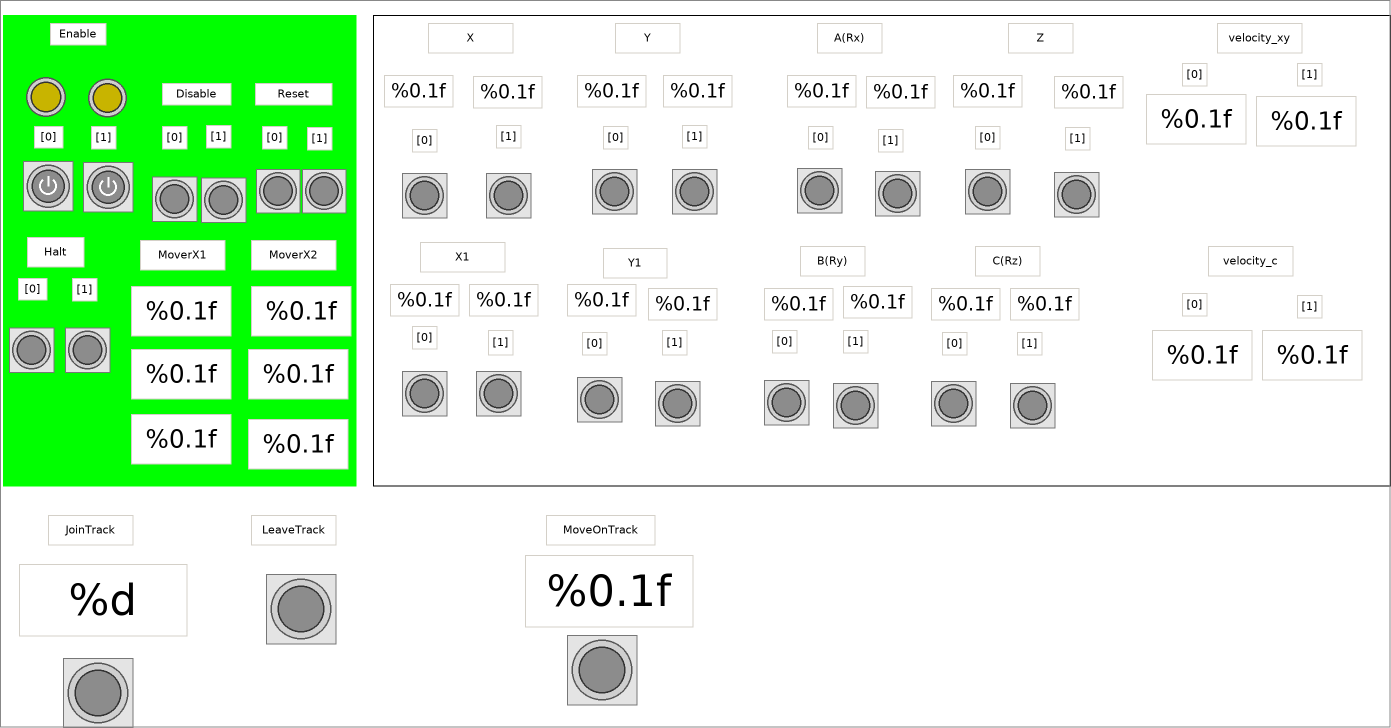
VISUALIZATION Visualization  // 1391x728
    Rectangle (373,15 1018x471)
    Rectangle (3,15 353x471)
    PowerSwitch (23,158 50x56), tooltip "Enable", variable: MAIN.enableM[0], behaviour: TOGGLE, style: Switch-PowerSwitch-Gray
    PushSwitch (152,159 45x80), tooltip "disable", variable: MAIN.disableM[0], behaviour: TAP, style: Switch-PushSwitch-Gray
    Lamp1 (23,64 46x66), variable: MAIN.Xpfeedback[0][0].Done, style: Lamp-Lamp1-Yellow
    PushSwitchLed (402,161 45x69), tooltip "movex", variable: MAIN.moveXM[0], behaviour: TOGGLE, style: Switch-PushSwitchLed-Gray
    Textfield (384,75 69x32), "%0.1f", text variable: MAIN.positionTargetX[0]
        OnMouseClick: write the text variable via Default, min 60, max 660
    Textfield (428,23 85x30), "X"
    Textfield (577,75 69x32), "%0.1f", text variable: MAIN.positionTargetY[0]
        OnMouseClick: write the text variable via Default, min 60, max 420
    Textfield (615,23 65x30), "Y"
    PushSwitchLed (592,160 45x63), tooltip "moveY", variable: MAIN.moveYM[0], behaviour: TOGGLE, style: Switch-PushSwitchLed-Gray
    Textfield (420,242 85x30), "X1"
    Textfield (603,248 64x30), "Y1"
    PushSwitchLed (402,359 45x69), tooltip "movex1", variable: MAIN.moveX1M[0], behaviour: TOGGLE, style: Switch-PushSwitchLed-Gray
    PushSwitchLed (577,365 45x69), tooltip "moveY1", variable: MAIN.moveY1M[0], behaviour: TOGGLE, style: Switch-PushSwitchLed-Gray
    Textfield (390,284 69x32), "%0.1f", text variable: MAIN.positionTargetX1[0]
        OnMouseClick: write the text variable via Default, min 60, max 660
    Textfield (567,284 69x32), "%0.1f", text variable: MAIN.positionTargetY1[0]
        OnMouseClick: write the text variable via Default, min 60, max 420
    Textfield (1146,94 100x50), "%0.1f", text variable: MAIN.velocity_xy[0]
        OnMouseClick: write the text variable via Default, min 1, max 2000
    Textfield (1217,23 85x30), "velocity_xy"
    Textfield (817,23 65x30), "A(Rx)"
    Textfield (787,75 69x32), "%0.1f", text variable: MAIN.positionTargetA[0]
        OnMouseClick: write the text variable via Default, min -5, max 5
    PushSwitchLed (797,159 45x63), tooltip "moveA", variable: MAIN.moveAM[0], behaviour: TOGGLE, style: Switch-PushSwitchLed-Gray
    Textfield (800,246 65x30), "B(Ry)"
    Textfield (764,288 69x32), "%0.1f", text variable: MAIN.positionTargetB[0]
        OnMouseClick: write the text variable via Default, min -5, max 5
    PushSwitchLed (764,368 45x69), tooltip "moveB", variable: MAIN.moveBM[0], behaviour: TOGGLE, style: Switch-PushSwitchLed-Gray
    Textfield (1008,23 65x30), "Z"
    Textfield (953,75 69x32), "%0.1f", text variable: MAIN.positionTargetZ[0]
        OnMouseClick: write the text variable via Default, min 2, max 5
    PushSwitchLed (965,160 45x63), tooltip "moveZ", variable: MAIN.moveZM[0], behaviour: TOGGLE, style: Switch-PushSwitchLed-Gray
    Textfield (975,246 65x30), "C(Rz)"
    Textfield (931,288 69x32), "%0.1f", text variable: MAIN.positionTargetC[0]
        OnMouseClick: write the text variable via Default
    PushSwitchLed (931,369 45x69), tooltip "moveC", variable: MAIN.moveCM[0], behaviour: TOGGLE, style: Switch-PushSwitchLed-Gray
    Textfield (1208,246 85x30), "velocity_c"
    Textfield (1152,330 100x50), "%0.1f", text variable: MAIN.velocity_c[0]
        OnMouseClick: write the text variable via Default, min 1, max 7000
    Textfield (131,286 100x50), "%0.1f", text variable: MAIN.Xpmover[0].MCTOPLC.ACT.ActPos.x
    Textfield (131,349 100x50), "%0.1f", text variable: MAIN.Xpmover[0].MCTOPLC.ACT.ActPos.y
    Textfield (131,414 100x50), "%0.1f", text variable: MAIN.Xpmover[0].MCTOPLC.ACT.ActPos.c
    Textfield (140,240 85x30), "MoverX1"
    PushSwitch (63,658 70x70), variable: MAIN.JoinTrack[0], behaviour: TOGGLE, style: Switch-PushSwitch-Gray
    PushSwitch (266,574 70x70), variable: MAIN.LeaveTrack[0], behaviour: TOGGLE, style: Switch-PushSwitch-Gray
    PushSwitch (567,635 70x70), variable: MAIN.MoveOnTrack[0], behaviour: TOGGLE, style: Switch-PushSwitch-Gray
    Textfield (48,515 85x30), "JoinTrack"
    Textfield (251,515 85x30), "LeaveTrack"
    Textfield (546,515 109x30), "MoveOnTrack"
    Textfield (19,564 168x72), "%d", text variable: MAIN.numberTrack[0]
        OnMouseClick: write the text variable via Default, min 0
    Textfield (525,555 168x72), "%0.1f", text variable: MAIN.distanceTrack[0]
        OnMouseClick: write the text variable via Default
    PushSwitch (256,160 44x62), variable: MAIN.ResetM[0], invisible if: MAIN.ResetM, behaviour: TOGGLE, style: Switch-PushSwitch-Gray
    Textfield (50,23 56x22), "Enable"
    Textfield (162,83 69x22), "Disable"
    Textfield (255,83 77x22), "Reset"
    PushSwitch (9,310 45x80), variable: MAIN.HaltM[0], invisible if: MAIN.HaltM, behaviour: TOGGLE, style: Switch-PushSwitch-Gray
    Textfield (27,237 57x30), "Halt"
    Textfield (34,126 29x22), "[0]"
    Textfield (91,126 25x23), "[1]"
    Lamp1 (85,66 45x64), variable: MAIN.Xpfeedback[1][0].Done, style: Lamp-Lamp1-Yellow
    PowerSwitch (83,159 50x56), tooltip "Enable", variable: MAIN.enableM[1], behaviour: TOGGLE, style: Switch-PowerSwitch-Gray
    Textfield (162,126 25x23), "[0]"
    Textfield (206,125 25x23), "[1]"
    PushSwitch (201,160 45x80), tooltip "disable", variable: MAIN.disableM[1], behaviour: TAP, style: Switch-PushSwitch-Gray
    Textfield (262,126 25x23), "[0]"
    PushSwitch (302,160 44x62), variable: MAIN.ResetM[1], invisible if: MAIN.ResetM, behaviour: TOGGLE, style: Switch-PushSwitch-Gray
    Textfield (307,127 25x23), "[1]"
    Textfield (496,125 25x23), "[1]"
    Textfield (412,129 25x23), "[0]"
    PushSwitchLed (486,161 45x69), tooltip "movex", variable: MAIN.moveXM[1], behaviour: TOGGLE, style: Switch-PushSwitchLed-Gray
    Textfield (603,126 25x23), "[0]"
    Textfield (473,76 69x32), "%0.1f", text variable: MAIN.positionTargetX[1]
        OnMouseClick: write the text variable via Default, min 60, max 660
    Textfield (663,75 69x32), "%0.1f", text variable: MAIN.positionTargetY[1]
        OnMouseClick: write the text variable via Default, min 60, max 420
    Textfield (682,125 25x23), "[1]"
    PushSwitchLed (672,160 45x63), tooltip "moveY", variable: MAIN.moveYM[1], behaviour: TOGGLE, style: Switch-PushSwitchLed-Gray
    Textfield (808,126 25x23), "[0]"
    Textfield (878,129 25x23), "[1]"
    Textfield (866,76 69x32), "%0.1f", text variable: MAIN.positionTargetA[1]
        OnMouseClick: write the text variable via Default, min -5, max 5
    PushSwitchLed (875,162 45x63), tooltip "moveA", variable: MAIN.moveAM[1], behaviour: TOGGLE, style: Switch-PushSwitchLed-Gray
    Textfield (975,126 25x23), "[0]"
    PushSwitchLed (1054,163 45x63), tooltip "moveZ", variable: MAIN.moveZM[1], behaviour: TOGGLE, style: Switch-PushSwitchLed-Gray
    Textfield (1065,127 25x23), "[1]"
    Textfield (1054,76 69x32), "%0.1f", text variable: MAIN.positionTargetZ[1]
        OnMouseClick: write the text variable via Default, min 2, max 5
    Textfield (412,326 25x23), "[0]"
    Textfield (469,284 69x32), "%0.1f", text variable: MAIN.positionTargetX1[1]
        OnMouseClick: write the text variable via Default, min 60, max 660
    Textfield (488,330 25x25), "[1]"
    PushSwitchLed (476,359 45x69), tooltip "movex1", variable: MAIN.moveX1M[1], behaviour: TOGGLE, style: Switch-PushSwitchLed-Gray
    Textfield (582,332 25x23), "[0]"
    Textfield (648,288 69x32), "%0.1f", text variable: MAIN.positionTargetY1[1]
        OnMouseClick: write the text variable via Default, min 60, max 420
    Textfield (662,330 25x25), "[1]"
    PushSwitchLed (655,369 45x69), tooltip "moveY1", variable: MAIN.moveY1M[1], behaviour: TOGGLE, style: Switch-PushSwitchLed-Gray
    Textfield (772,330 25x23), "[0]"
    PushSwitchLed (833,371 45x69), tooltip "moveB", variable: MAIN.moveBM[1], behaviour: TOGGLE, style: Switch-PushSwitchLed-Gray
    Textfield (843,286 69x32), "%0.1f", text variable: MAIN.positionTargetB[0]
        OnMouseClick: write the text variable via Default, min -5, max 5
    Textfield (843,330 25x23), "[1]"
    Textfield (942,332 25x23), "[0]"
    Textfield (1017,332 25x23), "[1]"
    Textfield (1010,288 69x32), "%0.1f", text variable: MAIN.positionTargetC[1]
        OnMouseClick: write the text variable via Default
    PushSwitchLed (1010,371 45x69), tooltip "moveC", variable: MAIN.moveCM[1], behaviour: TOGGLE, style: Switch-PushSwitchLed-Gray
    Textfield (1182,63 25x23), "[0]"
    Textfield (1256,96 100x50), "%0.1f", text variable: MAIN.velocity_xy[1]
        OnMouseClick: write the text variable via Default, min 1, max 2000
    Textfield (1297,63 25x23), "[1]"
    Textfield (1182,293 25x23), "[0]"
    Textfield (1297,295 25x23), "[1]"
    Textfield (1262,330 100x50), "%0.1f", text variable: MAIN.velocity_c[1]
        OnMouseClick: write the text variable via Default, min 1, max 7000
    Textfield (251,240 85x30), "MoverX2"
    Textfield (251,286 100x50), "%0.1f", text variable: MAIN.Xpmover[1].MCTOPLC.ACT.ActPos.x
    Textfield (248,349 100x50), "%0.1f", text variable: MAIN.Xpmover[1].MCTOPLC.ACT.ActPos.y
    Textfield (248,419 100x50), "%0.1f", text variable: MAIN.Xpmover[1].MCTOPLC.ACT.ActPos.c
    PushSwitch (65,310 45x80), variable: MAIN.HaltM[1], invisible if: MAIN.HaltM, behaviour: TOGGLE, style: Switch-PushSwitch-Gray
    Textfield (18,278 29x22), "[0]"
    Textfield (72,278 25x23), "[1]"
END_VISUALIZATION

(* stored: Version 1.1.0.1
   Visu Visualization: Id {c1681727-f998-4423-8310-7782445f4a53} *)
